(* Logix 5000 project; controller NSH_PLC2 vendor 1 type 14 code 167 rev 32.14; software revision 32.03; part 4 of 6 *)
(* tags used below, declared in another part *)
   AOI_MCC3_10J_ToPLC1 : E300ToMotor;
   AOI_MCC3_11A_ToPLC1 : E300ToMotor;
   AOI_MCC3_11D_ToPLC1 : E300ToMotor;
   AOI_MCC3_11G_ToPLC1 : E300ToMotor;
   AOI_MCC3_11J_ToPLC1 : E300ToMotor;
   AOI_MCC3_12A_ToPLC1 : E300ToMotor;
   AOI_MCC3_12C_ToPLC1 : E300ToMotor;
   AOI_MCC3_12E_ToPLC1 : E300ToMotor;
   AOI_MCC3_12G_ToPLC1 : E300ToMotor;
   AOI_MCC3_12J_ToPLC1 : E300ToMotor;
   AOI_MCC3_12L_ToPLC1 : E300ToMotor;
   AOI_MCC3_13A_ToPLC1 : E300ToMotor;
   AOI_MCC3_13C_ToPLC1 : E300ToMotor;
   AOI_MCC3_13E_ToPLC1 : E300ToMotor;
   AOI_MCC3_13G_ToPLC1 : E300ToMotor;
   AOI_MCC3_13J_ToPLC1 : E300ToMotor;
   AOI_MCC3_13L_ToPLC1 : E300ToMotor;
   AOI_MCC3_14A_ToPLC1 : E300ToMotor;
   AOI_MCC3_14C_ToPLC1 : E300ToMotor;
   AOI_MCC3_14E_ToPLC1 : E300ToMotor;
   AOI_MCC3_14G_ToPLC1 : E300ToMotor;
   AOI_MCC3_14J_ToPLC1 : E300ToMotor;
   AOI_MCC3_14L_ToPLC1 : E300ToMotor;
   AOI_MCC3_15A_ToPLC1 : E300ToMotor;
   AOI_MCC3_15C_ToPLC1 : E300ToMotor;
   AOI_MCC3_15E_ToPLC1 : E300ToMotor;
   AOI_MCC3_15G_ToPLC1 : E300ToMotor;
   AOI_MCC3_15J_ToPLC1 : E300ToMotor;
   AOI_MCC3_16A_ToPLC1 : E300ToMotor;
   AOI_MCC3_16C_ToPLC1 : E300ToMotor;
   AOI_MCC3_16E_ToPLC1 : E300ToMotor;
   AOI_MCC3_16G_ToPLC1 : E300ToMotor;
   AOI_MCC3_16J_ToPLC1 : E300ToMotor;
   AOI_MCC3_16L_ToPLC1 : E300ToMotor;
   AOI_MCC3_17A_ToPLC1 : E300ToMotor;
   AOI_MCC3_17C_ToPLC1 : E300ToMotor;
   AOI_MCC3_17E_ToPLC1 : E300ToMotor;
   AOI_MCC3_17G_ToPLC1 : E300ToMotor;
   AOI_MCC3_17J_ToPLC1 : E300ToMotor;
   AOI_MCC3_17L_ToPLC1 : E300ToMotor;
   AOI_MCC3_18A_ToPLC1 : E300ToMotor;
   AOI_MCC3_18C_ToPLC1 : E300ToMotor;
   AOI_MCC3_18E_ToPLC1 : E300ToMotor;
   AOI_MCC3_18G_ToPLC1 : E300ToMotor;
   AOI_MCC3_18J_ToPLC1 : E300ToMotor;
   AOI_MCC3_18L_ToPLC1 : E300ToMotor;
   AOI_MCC3_19A_ToPLC1 : E300ToMotor;
   AOI_MCC3_19C_ToPLC1 : E300ToMotor;
   AOI_MCC3_19E_ToPLC1 : E300ToMotor;
   AOI_MCC3_19G_ToPLC1 : E300ToMotor;
   AOI_MCC3_19J_ToPLC1 : E300ToMotor;
   AOI_MCC3_20A_ToPLC1 : E300ToMotor;
   AOI_MCC3_20C_ToPLC1 : E300ToMotor;
   AOI_MCC3_20E_ToPLC1 : E300ToMotor;
   AOI_MCC3_20G_ToPLC1 : E300ToMotor;
   AOI_MCC3_20J_ToPLC1 : E300ToMotor;
   AOI_MCC3_21A_ToPLC1 : E300ToMotor;
   AOI_MCC3_21C_ToPLC1 : E300ToMotor;
   AOI_MCC3_21E_ToPLC1 : E300ToMotor;
   AOI_MCC3_21G_ToPLC1 : E300ToMotor;
   AOI_MCC3_21J_ToPLC1 : E300ToMotor;
   AOI_MCC3_21L_ToPLC1 : E300ToMotor;
   AOI_MCC3_22C_ToPLC1 : E300ToMotor;
   AOI_MCC3_22E_ToPLC1 : E300ToMotor;
   AOI_MCC4_1E_ToPLC1 : PF525ToMotor;
   AOI_MCC4_2A_ToPLC1 : E300ToMotor;
   AOI_MCC4_2C_ToPLC1 : E300ToMotor;
   AOI_MCC4_2E_ToPLC1 : E300ToMotor;
   AOI_MCC4_2G_ToPLC1 : PF525ToMotor;
   AOI_MCC4_2K_ToPLC1 : PF525ToMotor;
   AOI_MCC4_3A_ToPLC1 : E300ToMotor;
   AOI_MCC4_3C_ToPLC1 : E300ToMotor;
   Const_4000_Hex : INT;   // Constant #16:4000, Entry Status Communicating
   GSV_EntryStatus : INT;   // GSV Entry Status, shold be #16:4000
   MCC3_10J_CommsOK : BOOL;   // Communications with AOP OK
   MCC3_11A_CommsOK : BOOL;   // Communications with AOP OK
   MCC3_11D_CommsOK : BOOL;   // Communications with AOP OK
   MCC3_11G_CommsOK : BOOL;   // Communications with AOP OK
   MCC3_11J_CommsOK : BOOL;   // Communications with AOP OK
   MCC3_12A_CommsOK : BOOL;   // Communications with AOP OK
   MCC3_12C_CommsOK : BOOL;   // Communications with AOP OK
   MCC3_12E_CommsOK : BOOL;   // Communications with AOP OK
   MCC3_12G_CommsOK : BOOL;   // Communications with AOP OK
   MCC3_12J_CommsOK : BOOL;   // Communications with AOP OK
   MCC3_12L_CommsOK : BOOL;   // Communications with AOP OK
   MCC3_13A_CommsOK : BOOL;   // Communications with AOP OK
   MCC3_13C_CommsOK : BOOL;   // Communications with AOP OK
   MCC3_13E_CommsOK : BOOL;   // Communications with AOP OK
   MCC3_13G_CommsOK : BOOL;   // Communications with AOP OK
   MCC3_13J_CommsOK : BOOL;   // Communications with AOP OK
   MCC3_13L_CommsOK : BOOL;   // Communications with AOP OK
   MCC3_14A_CommsOK : BOOL;   // Communications with AOP OK
   MCC3_14C_CommsOK : BOOL;   // Communications with AOP OK
   MCC3_14E_CommsOK : BOOL;   // Communications with AOP OK
   MCC3_14G_CommsOK : BOOL;   // Communications with AOP OK
   MCC3_14J_CommsOK : BOOL;   // Communications with AOP OK
   MCC3_14L_CommsOK : BOOL;   // Communications with AOP OK
   MCC3_15A_CommsOK : BOOL;   // Communications with AOP OK
   MCC3_15C_CommsOK : BOOL;   // Communications with AOP OK
   MCC3_15E_CommsOK : BOOL;   // Communications with AOP OK
   MCC3_15G_CommsOK : BOOL;   // Communications with AOP OK
   MCC3_15J_CommsOK : BOOL;   // Communications with AOP OK
   MCC3_16A_CommsOK : BOOL;   // Communications with AOP OK
   MCC3_16C_CommsOK : BOOL;   // Communications with AOP OK
   MCC3_16E_CommsOK : BOOL;   // Communications with AOP OK
   MCC3_16G_CommsOK : BOOL;   // Communications with AOP OK
   MCC3_16J_CommsOK : BOOL;   // Communications with AOP OK
   MCC3_16L_CommsOK : BOOL;   // Communications with AOP OK
   MCC3_17A_CommsOK : BOOL;   // Communications with AOP OK
   MCC3_17C_CommsOK : BOOL;   // Communications with AOP OK
   MCC3_17E_CommsOK : BOOL;   // Communications with AOP OK
   MCC3_17G_CommsOK : BOOL;   // Communications with AOP OK
   MCC3_17J_CommsOK : BOOL;   // Communications with AOP OK
   MCC3_17L_CommsOK : BOOL;   // Communications with AOP OK
   MCC3_18A_CommsOK : BOOL;   // Communications with AOP OK
   MCC3_18C_CommsOK : BOOL;   // Communications with AOP OK
   MCC3_18E_CommsOK : BOOL;   // Communications with AOP OK
   MCC3_18G_CommsOK : BOOL;   // Communications with AOP OK
   MCC3_18J_CommsOK : BOOL;   // Communications with AOP OK
   MCC3_18L_CommsOK : BOOL;   // Communications with AOP OK
   MCC3_19A_CommsOK : BOOL;   // Communications with AOP OK
   MCC3_19C_CommsOK : BOOL;   // Communications with AOP OK
   MCC3_19E_CommsOK : BOOL;   // Communications with AOP OK
   MCC3_19G_CommsOK : BOOL;   // Communications with AOP OK
   MCC3_19J_CommsOK : BOOL;   // Communications with AOP OK
   MCC3_20A_CommsOK : BOOL;   // Communications with AOP OK
   MCC3_20C_CommsOK : BOOL;   // Communications with AOP OK
   MCC3_20E_CommsOK : BOOL;   // Communications with AOP OK
   MCC3_20G_CommsOK : BOOL;   // Communications with AOP OK
   MCC3_20J_CommsOK : BOOL;   // Communications with AOP OK
   MCC3_21A_CommsOK : BOOL;   // Communications with AOP OK
   MCC3_21C_CommsOK : BOOL;   // Communications with AOP OK
   MCC3_21E_CommsOK : BOOL;   // Communications with AOP OK
   MCC3_21G_CommsOK : BOOL;   // Communications with AOP OK
   MCC3_21J_CommsOK : BOOL;   // Communications with AOP OK
   MCC3_21L_CommsOK : BOOL;   // Communications with AOP OK
   MCC3_22C_CommsOK : BOOL;   // Communications with AOP OK
   MCC3_22E_CommsOK : BOOL;   // Communications with AOP OK
   MCC4_1E_CommsOK : BOOL;   // Communications with AOP OK
   MCC4_2A_CommsOK : BOOL;   // Communications with AOP OK
   MCC4_2C_CommsOK : BOOL;   // Communications with AOP OK
   MCC4_2E_CommsOK : BOOL;   // Communications with AOP OK
   MCC4_2G_CommsOK : BOOL;   // Communications with AOP OK
   MCC4_2K_CommsOK : BOOL;   // Communications with AOP OK
   MCC4_3A_CommsOK : BOOL;   // Communications with AOP OK
   MCC4_3C_CommsOK : BOOL;   // Communications with AOP OK
   MotorsStatusTag : MotorsStatusUDT;   // Only Instance of UDT
(* MainProgram, continued *)

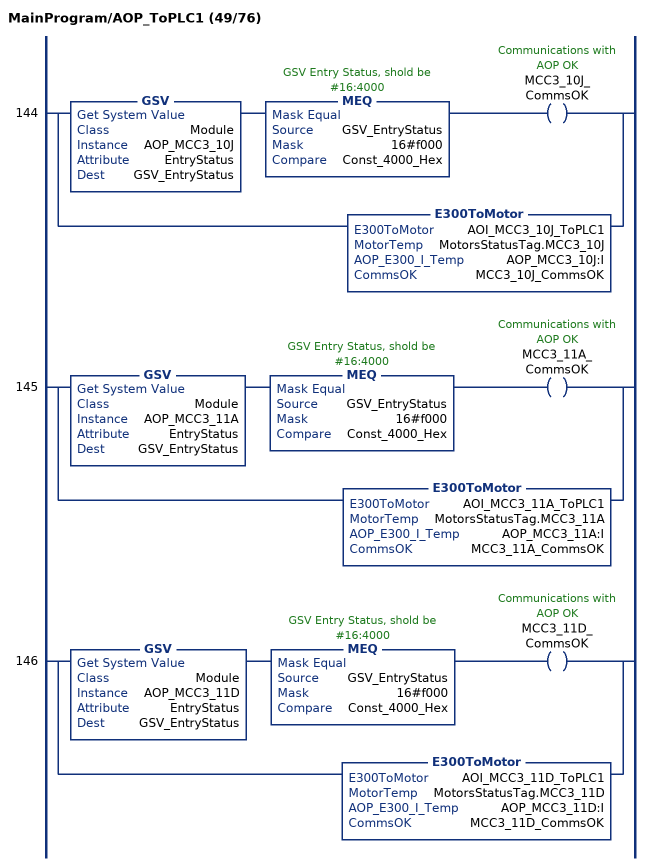
   [picture p55: MainProgram/AOP_ToPLC1 rungs 144-146]
   144: [GSV(Module,AOP_MCC3_10J,EntryStatus,GSV_EntryStatus) MEQ(GSV_EntryStatus,16#f000,Const_4000_Hex) OTE(MCC3_10J_CommsOK) ,E300ToMotor(AOI_MCC3_10J_ToPLC1,MotorsStatusTag.MCC3_10J,AOP_MCC3_10J:I,MCC3_10J_CommsOK) ];
   145: [GSV(Module,AOP_MCC3_11A,EntryStatus,GSV_EntryStatus) MEQ(GSV_EntryStatus,16#f000,Const_4000_Hex) OTE(MCC3_11A_CommsOK) ,E300ToMotor(AOI_MCC3_11A_ToPLC1,MotorsStatusTag.MCC3_11A,AOP_MCC3_11A:I,MCC3_11A_CommsOK) ];
   146: [GSV(Module,AOP_MCC3_11D,EntryStatus,GSV_EntryStatus) MEQ(GSV_EntryStatus,16#f000,Const_4000_Hex) OTE(MCC3_11D_CommsOK) ,E300ToMotor(AOI_MCC3_11D_ToPLC1,MotorsStatusTag.MCC3_11D,AOP_MCC3_11D:I,MCC3_11D_CommsOK) ];
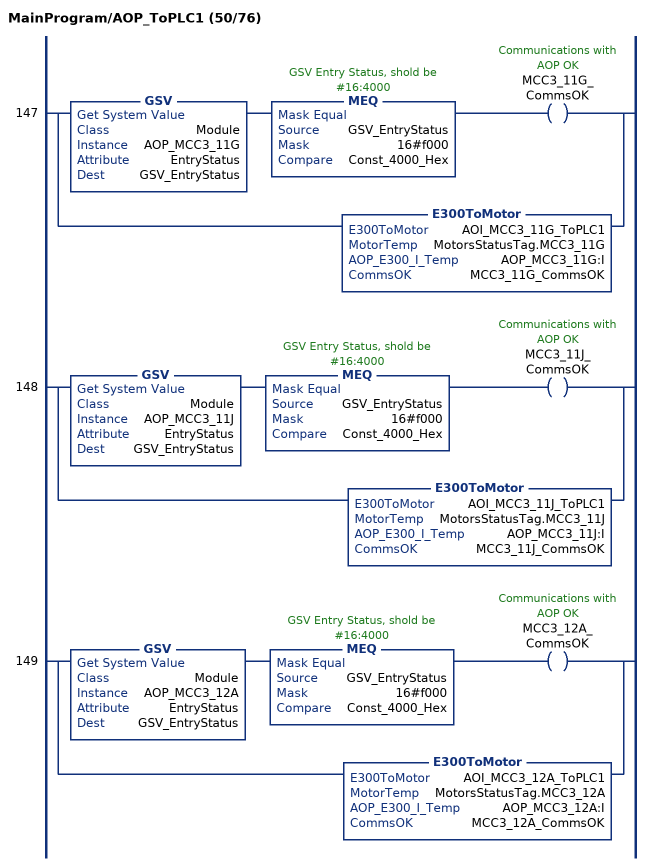
   147: [GSV(Module,AOP_MCC3_11G,EntryStatus,GSV_EntryStatus) MEQ(GSV_EntryStatus,16#f000,Const_4000_Hex) OTE(MCC3_11G_CommsOK) ,E300ToMotor(AOI_MCC3_11G_ToPLC1,MotorsStatusTag.MCC3_11G,AOP_MCC3_11G:I,MCC3_11G_CommsOK) ];
   148: [GSV(Module,AOP_MCC3_11J,EntryStatus,GSV_EntryStatus) MEQ(GSV_EntryStatus,16#f000,Const_4000_Hex) OTE(MCC3_11J_CommsOK) ,E300ToMotor(AOI_MCC3_11J_ToPLC1,MotorsStatusTag.MCC3_11J,AOP_MCC3_11J:I,MCC3_11J_CommsOK) ];
   149: [GSV(Module,AOP_MCC3_12A,EntryStatus,GSV_EntryStatus) MEQ(GSV_EntryStatus,16#f000,Const_4000_Hex) OTE(MCC3_12A_CommsOK) ,E300ToMotor(AOI_MCC3_12A_ToPLC1,MotorsStatusTag.MCC3_12A,AOP_MCC3_12A:I,MCC3_12A_CommsOK) ];
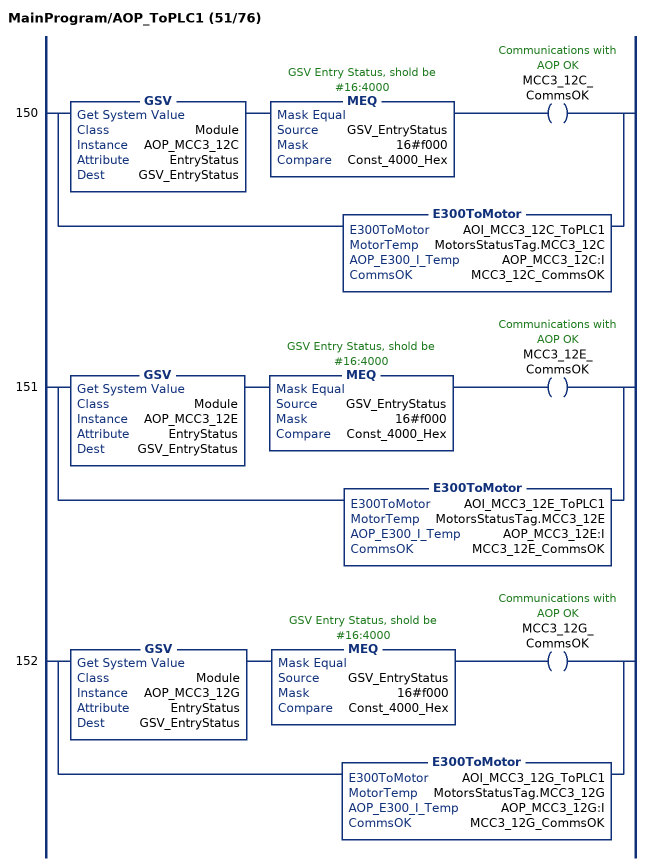
   150: [GSV(Module,AOP_MCC3_12C,EntryStatus,GSV_EntryStatus) MEQ(GSV_EntryStatus,16#f000,Const_4000_Hex) OTE(MCC3_12C_CommsOK) ,E300ToMotor(AOI_MCC3_12C_ToPLC1,MotorsStatusTag.MCC3_12C,AOP_MCC3_12C:I,MCC3_12C_CommsOK) ];
   151: [GSV(Module,AOP_MCC3_12E,EntryStatus,GSV_EntryStatus) MEQ(GSV_EntryStatus,16#f000,Const_4000_Hex) OTE(MCC3_12E_CommsOK) ,E300ToMotor(AOI_MCC3_12E_ToPLC1,MotorsStatusTag.MCC3_12E,AOP_MCC3_12E:I,MCC3_12E_CommsOK) ];
   152: [GSV(Module,AOP_MCC3_12G,EntryStatus,GSV_EntryStatus) MEQ(GSV_EntryStatus,16#f000,Const_4000_Hex) OTE(MCC3_12G_CommsOK) ,E300ToMotor(AOI_MCC3_12G_ToPLC1,MotorsStatusTag.MCC3_12G,AOP_MCC3_12G:I,MCC3_12G_CommsOK) ];
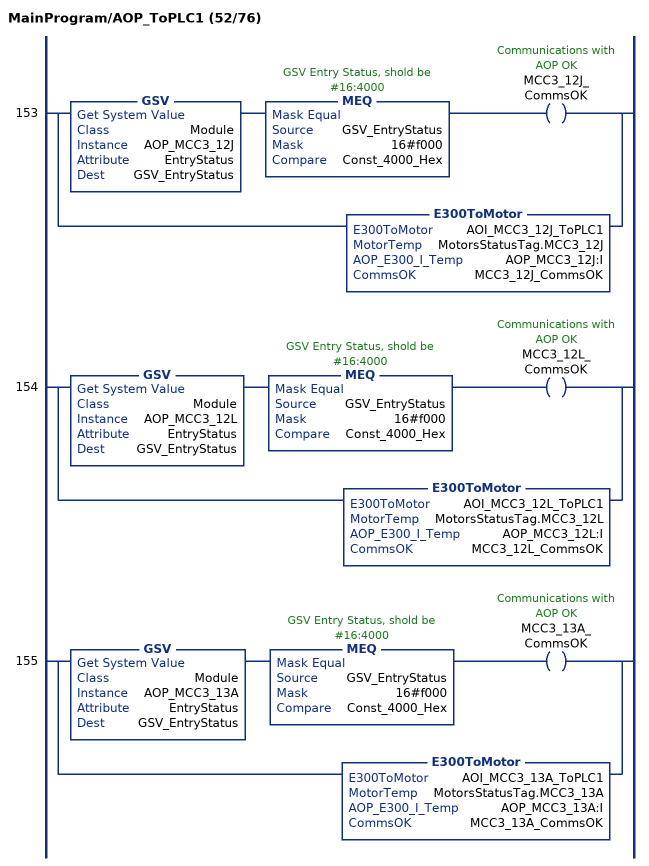
   153: [GSV(Module,AOP_MCC3_12J,EntryStatus,GSV_EntryStatus) MEQ(GSV_EntryStatus,16#f000,Const_4000_Hex) OTE(MCC3_12J_CommsOK) ,E300ToMotor(AOI_MCC3_12J_ToPLC1,MotorsStatusTag.MCC3_12J,AOP_MCC3_12J:I,MCC3_12J_CommsOK) ];
   154: [GSV(Module,AOP_MCC3_12L,EntryStatus,GSV_EntryStatus) MEQ(GSV_EntryStatus,16#f000,Const_4000_Hex) OTE(MCC3_12L_CommsOK) ,E300ToMotor(AOI_MCC3_12L_ToPLC1,MotorsStatusTag.MCC3_12L,AOP_MCC3_12L:I,MCC3_12L_CommsOK) ];
   155: [GSV(Module,AOP_MCC3_13A,EntryStatus,GSV_EntryStatus) MEQ(GSV_EntryStatus,16#f000,Const_4000_Hex) OTE(MCC3_13A_CommsOK) ,E300ToMotor(AOI_MCC3_13A_ToPLC1,MotorsStatusTag.MCC3_13A,AOP_MCC3_13A:I,MCC3_13A_CommsOK) ];
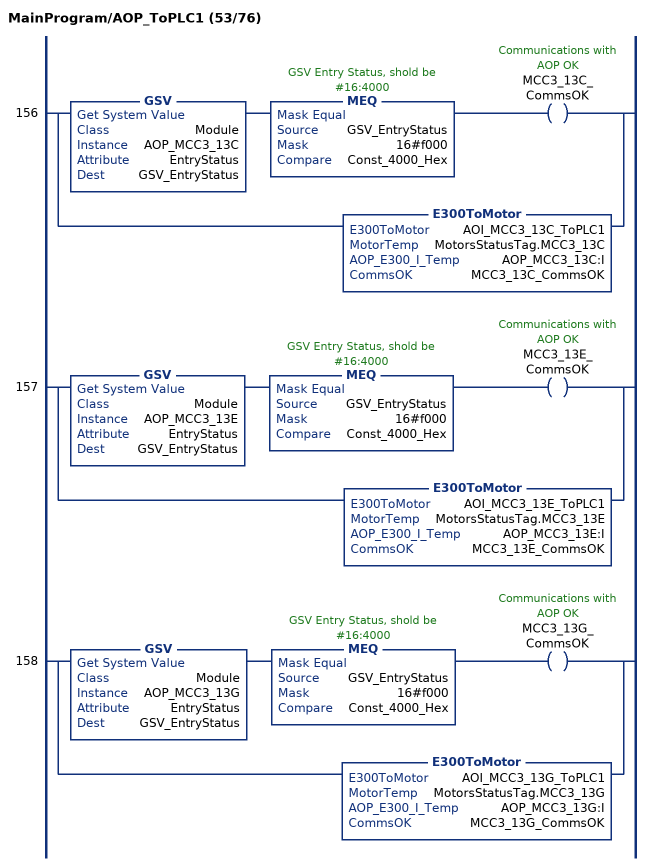
   156: [GSV(Module,AOP_MCC3_13C,EntryStatus,GSV_EntryStatus) MEQ(GSV_EntryStatus,16#f000,Const_4000_Hex) OTE(MCC3_13C_CommsOK) ,E300ToMotor(AOI_MCC3_13C_ToPLC1,MotorsStatusTag.MCC3_13C,AOP_MCC3_13C:I,MCC3_13C_CommsOK) ];
   157: [GSV(Module,AOP_MCC3_13E,EntryStatus,GSV_EntryStatus) MEQ(GSV_EntryStatus,16#f000,Const_4000_Hex) OTE(MCC3_13E_CommsOK) ,E300ToMotor(AOI_MCC3_13E_ToPLC1,MotorsStatusTag.MCC3_13E,AOP_MCC3_13E:I,MCC3_13E_CommsOK) ];
   158: [GSV(Module,AOP_MCC3_13G,EntryStatus,GSV_EntryStatus) MEQ(GSV_EntryStatus,16#f000,Const_4000_Hex) OTE(MCC3_13G_CommsOK) ,E300ToMotor(AOI_MCC3_13G_ToPLC1,MotorsStatusTag.MCC3_13G,AOP_MCC3_13G:I,MCC3_13G_CommsOK) ];
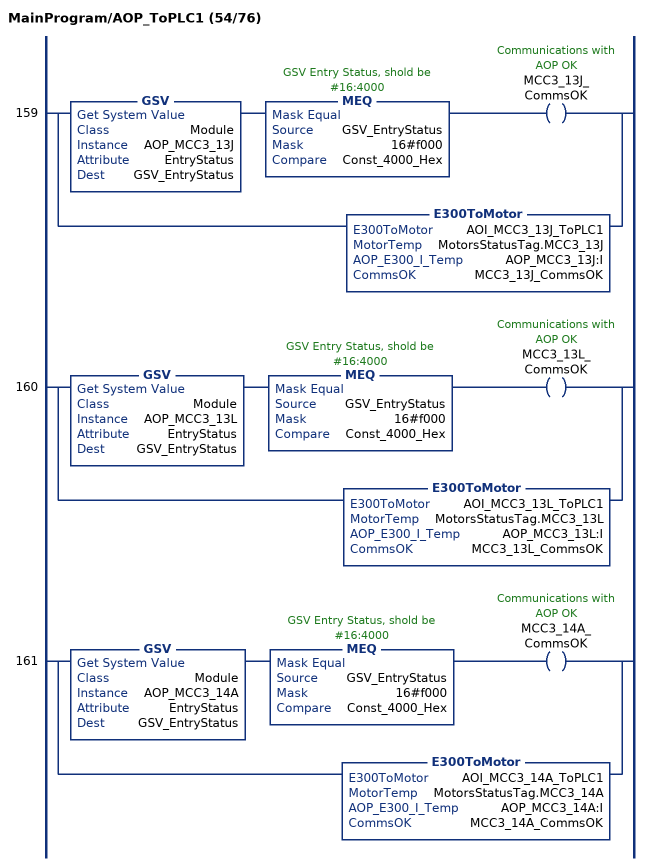
   159: [GSV(Module,AOP_MCC3_13J,EntryStatus,GSV_EntryStatus) MEQ(GSV_EntryStatus,16#f000,Const_4000_Hex) OTE(MCC3_13J_CommsOK) ,E300ToMotor(AOI_MCC3_13J_ToPLC1,MotorsStatusTag.MCC3_13J,AOP_MCC3_13J:I,MCC3_13J_CommsOK) ];
   160: [GSV(Module,AOP_MCC3_13L,EntryStatus,GSV_EntryStatus) MEQ(GSV_EntryStatus,16#f000,Const_4000_Hex) OTE(MCC3_13L_CommsOK) ,E300ToMotor(AOI_MCC3_13L_ToPLC1,MotorsStatusTag.MCC3_13L,AOP_MCC3_13L:I,MCC3_13L_CommsOK) ];
   161: [GSV(Module,AOP_MCC3_14A,EntryStatus,GSV_EntryStatus) MEQ(GSV_EntryStatus,16#f000,Const_4000_Hex) OTE(MCC3_14A_CommsOK) ,E300ToMotor(AOI_MCC3_14A_ToPLC1,MotorsStatusTag.MCC3_14A,AOP_MCC3_14A:I,MCC3_14A_CommsOK) ];
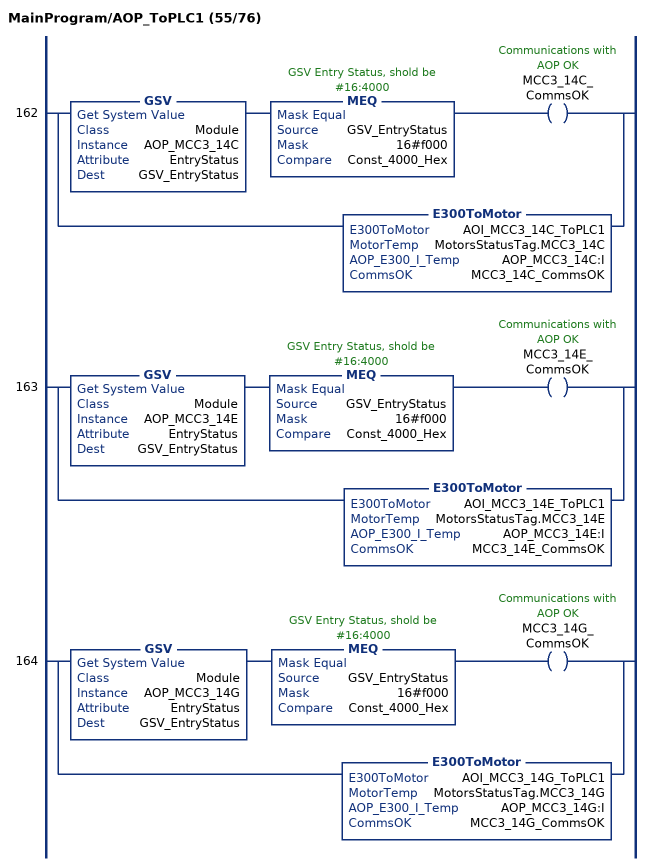
   162: [GSV(Module,AOP_MCC3_14C,EntryStatus,GSV_EntryStatus) MEQ(GSV_EntryStatus,16#f000,Const_4000_Hex) OTE(MCC3_14C_CommsOK) ,E300ToMotor(AOI_MCC3_14C_ToPLC1,MotorsStatusTag.MCC3_14C,AOP_MCC3_14C:I,MCC3_14C_CommsOK) ];
   163: [GSV(Module,AOP_MCC3_14E,EntryStatus,GSV_EntryStatus) MEQ(GSV_EntryStatus,16#f000,Const_4000_Hex) OTE(MCC3_14E_CommsOK) ,E300ToMotor(AOI_MCC3_14E_ToPLC1,MotorsStatusTag.MCC3_14E,AOP_MCC3_14E:I,MCC3_14E_CommsOK) ];
   164: [GSV(Module,AOP_MCC3_14G,EntryStatus,GSV_EntryStatus) MEQ(GSV_EntryStatus,16#f000,Const_4000_Hex) OTE(MCC3_14G_CommsOK) ,E300ToMotor(AOI_MCC3_14G_ToPLC1,MotorsStatusTag.MCC3_14G,AOP_MCC3_14G:I,MCC3_14G_CommsOK) ];
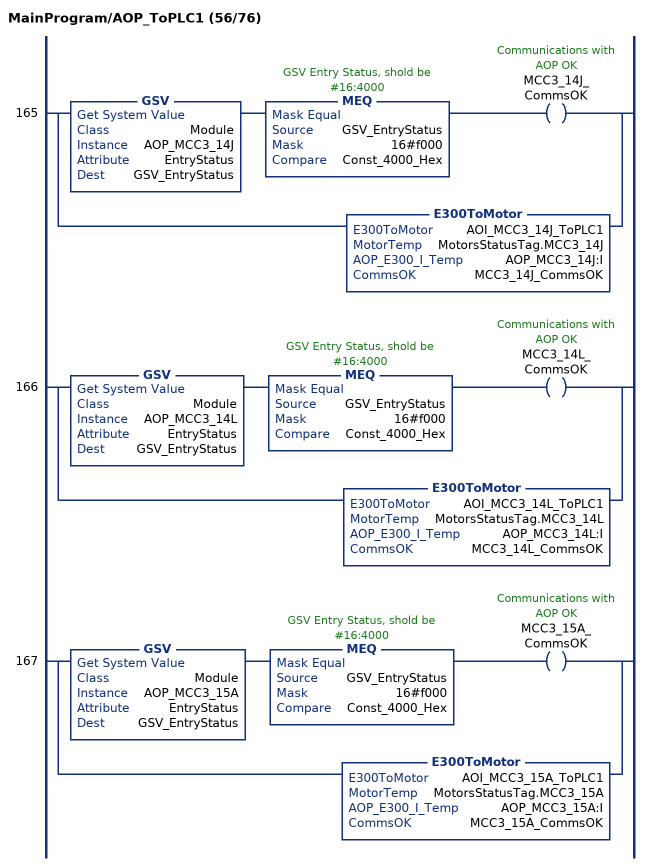
   165: [GSV(Module,AOP_MCC3_14J,EntryStatus,GSV_EntryStatus) MEQ(GSV_EntryStatus,16#f000,Const_4000_Hex) OTE(MCC3_14J_CommsOK) ,E300ToMotor(AOI_MCC3_14J_ToPLC1,MotorsStatusTag.MCC3_14J,AOP_MCC3_14J:I,MCC3_14J_CommsOK) ];
   166: [GSV(Module,AOP_MCC3_14L,EntryStatus,GSV_EntryStatus) MEQ(GSV_EntryStatus,16#f000,Const_4000_Hex) OTE(MCC3_14L_CommsOK) ,E300ToMotor(AOI_MCC3_14L_ToPLC1,MotorsStatusTag.MCC3_14L,AOP_MCC3_14L:I,MCC3_14L_CommsOK) ];
   167: [GSV(Module,AOP_MCC3_15A,EntryStatus,GSV_EntryStatus) MEQ(GSV_EntryStatus,16#f000,Const_4000_Hex) OTE(MCC3_15A_CommsOK) ,E300ToMotor(AOI_MCC3_15A_ToPLC1,MotorsStatusTag.MCC3_15A,AOP_MCC3_15A:I,MCC3_15A_CommsOK) ];
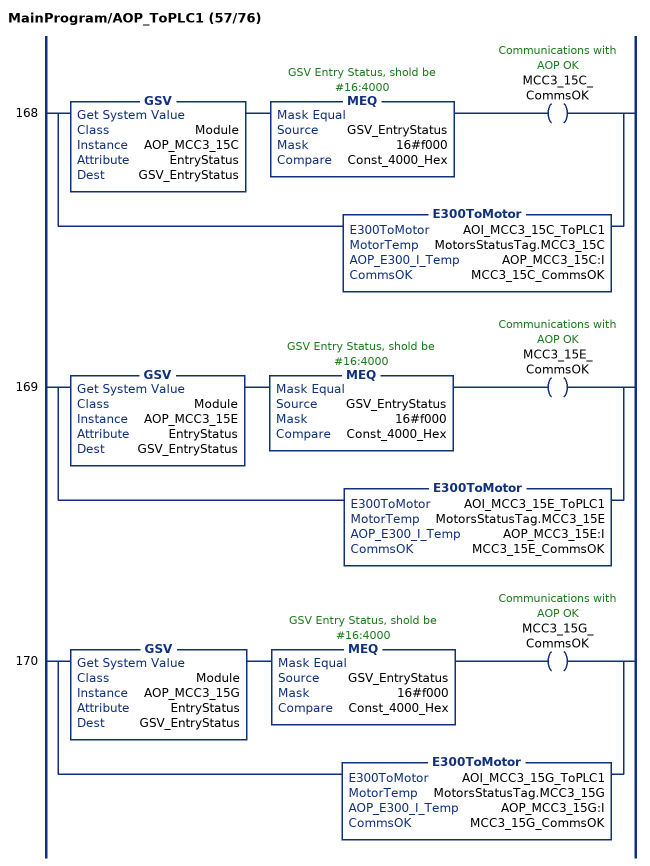
   168: [GSV(Module,AOP_MCC3_15C,EntryStatus,GSV_EntryStatus) MEQ(GSV_EntryStatus,16#f000,Const_4000_Hex) OTE(MCC3_15C_CommsOK) ,E300ToMotor(AOI_MCC3_15C_ToPLC1,MotorsStatusTag.MCC3_15C,AOP_MCC3_15C:I,MCC3_15C_CommsOK) ];
   169: [GSV(Module,AOP_MCC3_15E,EntryStatus,GSV_EntryStatus) MEQ(GSV_EntryStatus,16#f000,Const_4000_Hex) OTE(MCC3_15E_CommsOK) ,E300ToMotor(AOI_MCC3_15E_ToPLC1,MotorsStatusTag.MCC3_15E,AOP_MCC3_15E:I,MCC3_15E_CommsOK) ];
   170: [GSV(Module,AOP_MCC3_15G,EntryStatus,GSV_EntryStatus) MEQ(GSV_EntryStatus,16#f000,Const_4000_Hex) OTE(MCC3_15G_CommsOK) ,E300ToMotor(AOI_MCC3_15G_ToPLC1,MotorsStatusTag.MCC3_15G,AOP_MCC3_15G:I,MCC3_15G_CommsOK) ];
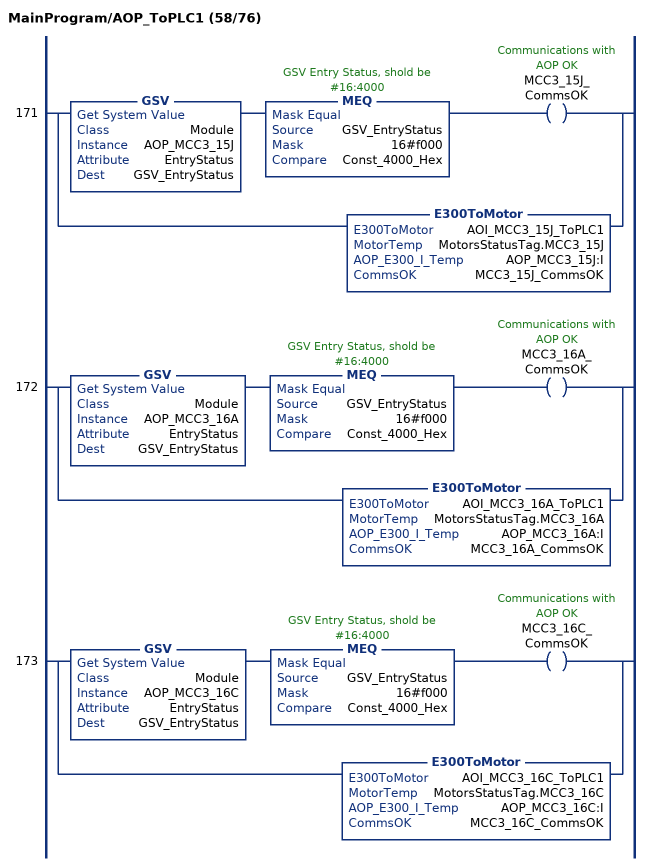
   171: [GSV(Module,AOP_MCC3_15J,EntryStatus,GSV_EntryStatus) MEQ(GSV_EntryStatus,16#f000,Const_4000_Hex) OTE(MCC3_15J_CommsOK) ,E300ToMotor(AOI_MCC3_15J_ToPLC1,MotorsStatusTag.MCC3_15J,AOP_MCC3_15J:I,MCC3_15J_CommsOK) ];
   172: [GSV(Module,AOP_MCC3_16A,EntryStatus,GSV_EntryStatus) MEQ(GSV_EntryStatus,16#f000,Const_4000_Hex) OTE(MCC3_16A_CommsOK) ,E300ToMotor(AOI_MCC3_16A_ToPLC1,MotorsStatusTag.MCC3_16A,AOP_MCC3_16A:I,MCC3_16A_CommsOK) ];
   173: [GSV(Module,AOP_MCC3_16C,EntryStatus,GSV_EntryStatus) MEQ(GSV_EntryStatus,16#f000,Const_4000_Hex) OTE(MCC3_16C_CommsOK) ,E300ToMotor(AOI_MCC3_16C_ToPLC1,MotorsStatusTag.MCC3_16C,AOP_MCC3_16C:I,MCC3_16C_CommsOK) ];
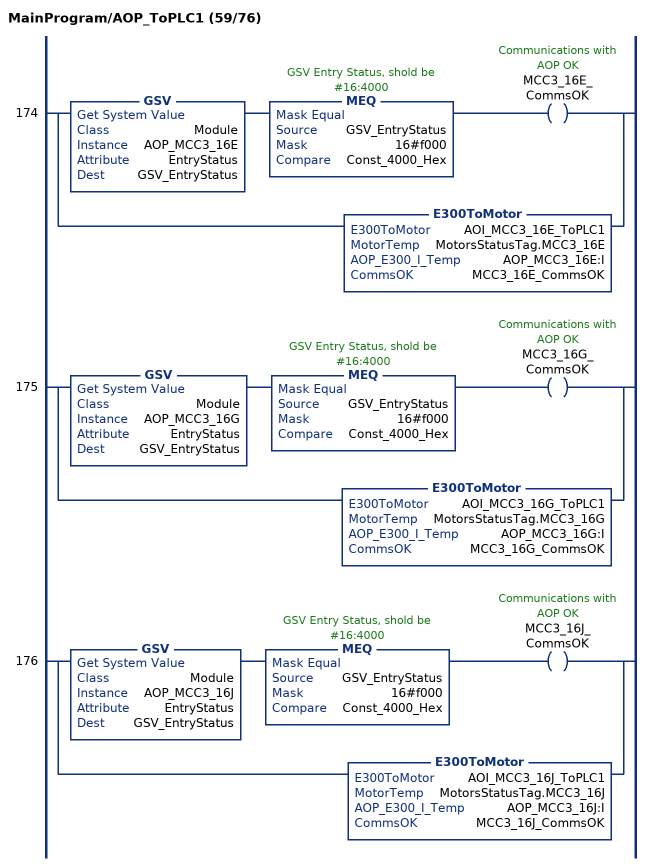
   174: [GSV(Module,AOP_MCC3_16E,EntryStatus,GSV_EntryStatus) MEQ(GSV_EntryStatus,16#f000,Const_4000_Hex) OTE(MCC3_16E_CommsOK) ,E300ToMotor(AOI_MCC3_16E_ToPLC1,MotorsStatusTag.MCC3_16E,AOP_MCC3_16E:I,MCC3_16E_CommsOK) ];
   175: [GSV(Module,AOP_MCC3_16G,EntryStatus,GSV_EntryStatus) MEQ(GSV_EntryStatus,16#f000,Const_4000_Hex) OTE(MCC3_16G_CommsOK) ,E300ToMotor(AOI_MCC3_16G_ToPLC1,MotorsStatusTag.MCC3_16G,AOP_MCC3_16G:I,MCC3_16G_CommsOK) ];
   176: [GSV(Module,AOP_MCC3_16J,EntryStatus,GSV_EntryStatus) MEQ(GSV_EntryStatus,16#f000,Const_4000_Hex) OTE(MCC3_16J_CommsOK) ,E300ToMotor(AOI_MCC3_16J_ToPLC1,MotorsStatusTag.MCC3_16J,AOP_MCC3_16J:I,MCC3_16J_CommsOK) ];
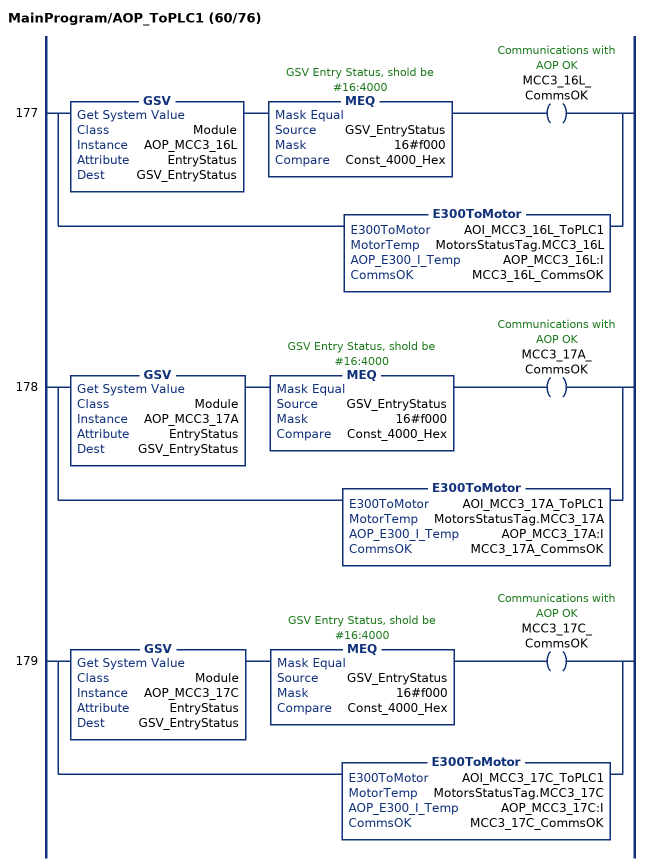
   177: [GSV(Module,AOP_MCC3_16L,EntryStatus,GSV_EntryStatus) MEQ(GSV_EntryStatus,16#f000,Const_4000_Hex) OTE(MCC3_16L_CommsOK) ,E300ToMotor(AOI_MCC3_16L_ToPLC1,MotorsStatusTag.MCC3_16L,AOP_MCC3_16L:I,MCC3_16L_CommsOK) ];
   178: [GSV(Module,AOP_MCC3_17A,EntryStatus,GSV_EntryStatus) MEQ(GSV_EntryStatus,16#f000,Const_4000_Hex) OTE(MCC3_17A_CommsOK) ,E300ToMotor(AOI_MCC3_17A_ToPLC1,MotorsStatusTag.MCC3_17A,AOP_MCC3_17A:I,MCC3_17A_CommsOK) ];
   179: [GSV(Module,AOP_MCC3_17C,EntryStatus,GSV_EntryStatus) MEQ(GSV_EntryStatus,16#f000,Const_4000_Hex) OTE(MCC3_17C_CommsOK) ,E300ToMotor(AOI_MCC3_17C_ToPLC1,MotorsStatusTag.MCC3_17C,AOP_MCC3_17C:I,MCC3_17C_CommsOK) ];
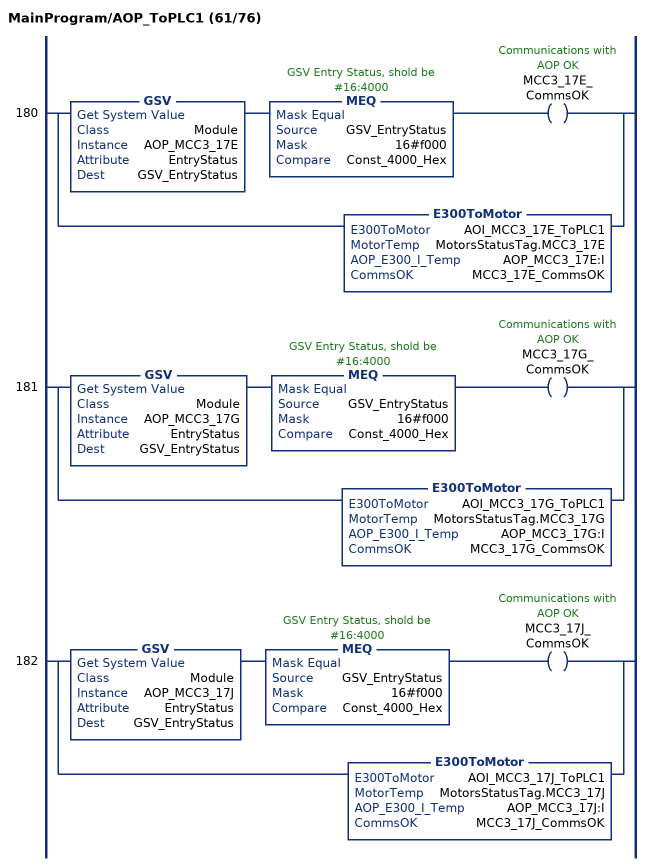
   180: [GSV(Module,AOP_MCC3_17E,EntryStatus,GSV_EntryStatus) MEQ(GSV_EntryStatus,16#f000,Const_4000_Hex) OTE(MCC3_17E_CommsOK) ,E300ToMotor(AOI_MCC3_17E_ToPLC1,MotorsStatusTag.MCC3_17E,AOP_MCC3_17E:I,MCC3_17E_CommsOK) ];
   181: [GSV(Module,AOP_MCC3_17G,EntryStatus,GSV_EntryStatus) MEQ(GSV_EntryStatus,16#f000,Const_4000_Hex) OTE(MCC3_17G_CommsOK) ,E300ToMotor(AOI_MCC3_17G_ToPLC1,MotorsStatusTag.MCC3_17G,AOP_MCC3_17G:I,MCC3_17G_CommsOK) ];
   182: [GSV(Module,AOP_MCC3_17J,EntryStatus,GSV_EntryStatus) MEQ(GSV_EntryStatus,16#f000,Const_4000_Hex) OTE(MCC3_17J_CommsOK) ,E300ToMotor(AOI_MCC3_17J_ToPLC1,MotorsStatusTag.MCC3_17J,AOP_MCC3_17J:I,MCC3_17J_CommsOK) ];
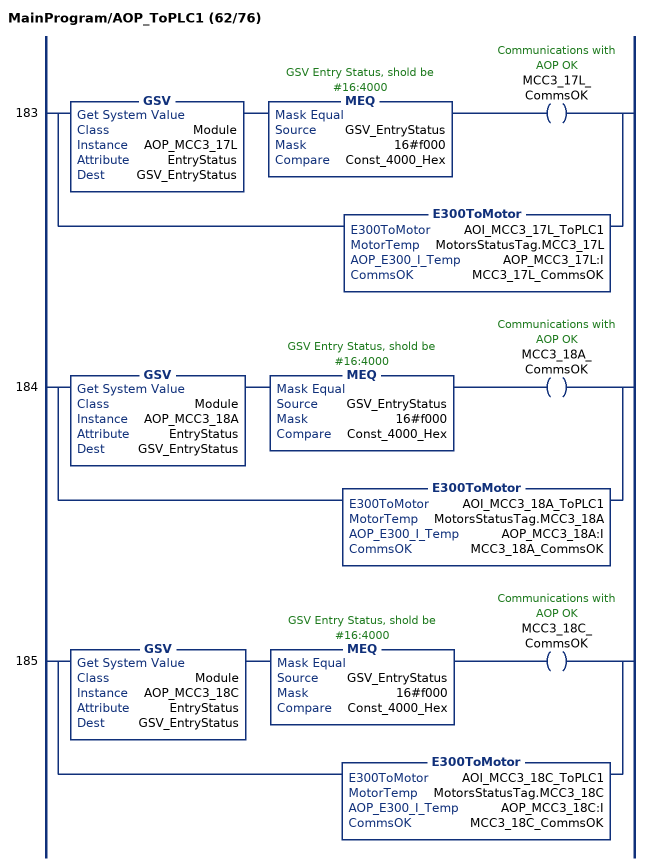
   183: [GSV(Module,AOP_MCC3_17L,EntryStatus,GSV_EntryStatus) MEQ(GSV_EntryStatus,16#f000,Const_4000_Hex) OTE(MCC3_17L_CommsOK) ,E300ToMotor(AOI_MCC3_17L_ToPLC1,MotorsStatusTag.MCC3_17L,AOP_MCC3_17L:I,MCC3_17L_CommsOK) ];
   184: [GSV(Module,AOP_MCC3_18A,EntryStatus,GSV_EntryStatus) MEQ(GSV_EntryStatus,16#f000,Const_4000_Hex) OTE(MCC3_18A_CommsOK) ,E300ToMotor(AOI_MCC3_18A_ToPLC1,MotorsStatusTag.MCC3_18A,AOP_MCC3_18A:I,MCC3_18A_CommsOK) ];
   185: [GSV(Module,AOP_MCC3_18C,EntryStatus,GSV_EntryStatus) MEQ(GSV_EntryStatus,16#f000,Const_4000_Hex) OTE(MCC3_18C_CommsOK) ,E300ToMotor(AOI_MCC3_18C_ToPLC1,MotorsStatusTag.MCC3_18C,AOP_MCC3_18C:I,MCC3_18C_CommsOK) ];
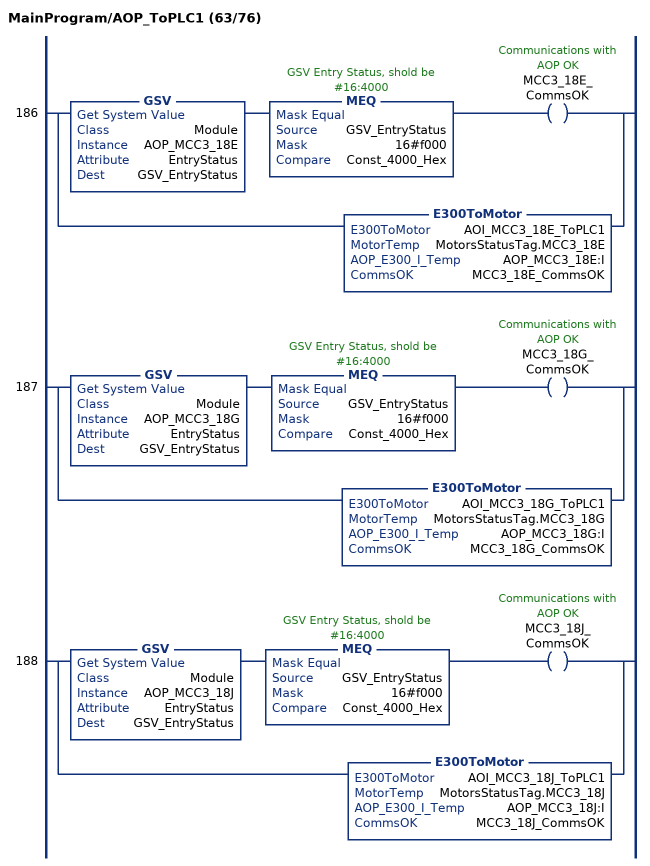
   186: [GSV(Module,AOP_MCC3_18E,EntryStatus,GSV_EntryStatus) MEQ(GSV_EntryStatus,16#f000,Const_4000_Hex) OTE(MCC3_18E_CommsOK) ,E300ToMotor(AOI_MCC3_18E_ToPLC1,MotorsStatusTag.MCC3_18E,AOP_MCC3_18E:I,MCC3_18E_CommsOK) ];
   187: [GSV(Module,AOP_MCC3_18G,EntryStatus,GSV_EntryStatus) MEQ(GSV_EntryStatus,16#f000,Const_4000_Hex) OTE(MCC3_18G_CommsOK) ,E300ToMotor(AOI_MCC3_18G_ToPLC1,MotorsStatusTag.MCC3_18G,AOP_MCC3_18G:I,MCC3_18G_CommsOK) ];
   188: [GSV(Module,AOP_MCC3_18J,EntryStatus,GSV_EntryStatus) MEQ(GSV_EntryStatus,16#f000,Const_4000_Hex) OTE(MCC3_18J_CommsOK) ,E300ToMotor(AOI_MCC3_18J_ToPLC1,MotorsStatusTag.MCC3_18J,AOP_MCC3_18J:I,MCC3_18J_CommsOK) ];
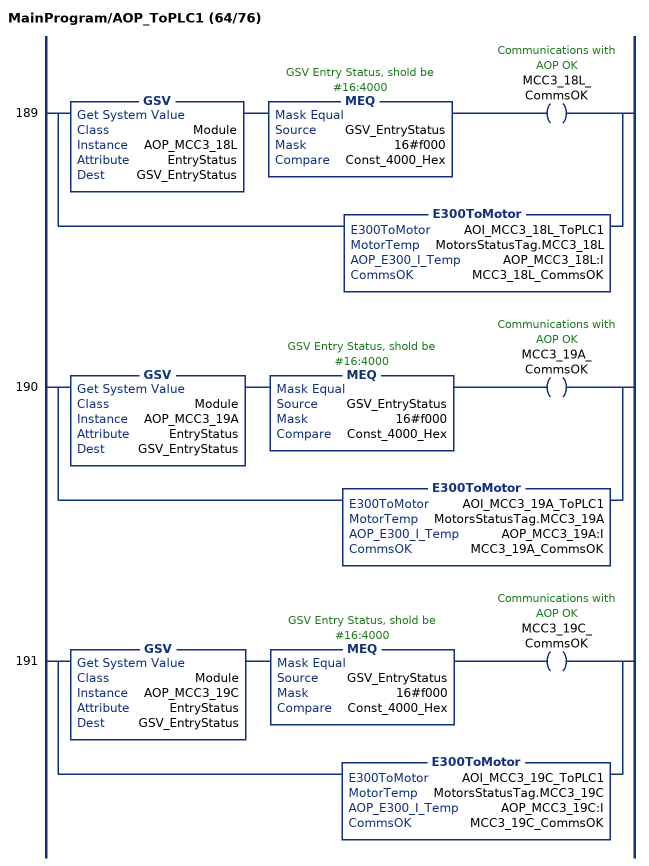
   189: [GSV(Module,AOP_MCC3_18L,EntryStatus,GSV_EntryStatus) MEQ(GSV_EntryStatus,16#f000,Const_4000_Hex) OTE(MCC3_18L_CommsOK) ,E300ToMotor(AOI_MCC3_18L_ToPLC1,MotorsStatusTag.MCC3_18L,AOP_MCC3_18L:I,MCC3_18L_CommsOK) ];
   190: [GSV(Module,AOP_MCC3_19A,EntryStatus,GSV_EntryStatus) MEQ(GSV_EntryStatus,16#f000,Const_4000_Hex) OTE(MCC3_19A_CommsOK) ,E300ToMotor(AOI_MCC3_19A_ToPLC1,MotorsStatusTag.MCC3_19A,AOP_MCC3_19A:I,MCC3_19A_CommsOK) ];
   191: [GSV(Module,AOP_MCC3_19C,EntryStatus,GSV_EntryStatus) MEQ(GSV_EntryStatus,16#f000,Const_4000_Hex) OTE(MCC3_19C_CommsOK) ,E300ToMotor(AOI_MCC3_19C_ToPLC1,MotorsStatusTag.MCC3_19C,AOP_MCC3_19C:I,MCC3_19C_CommsOK) ];
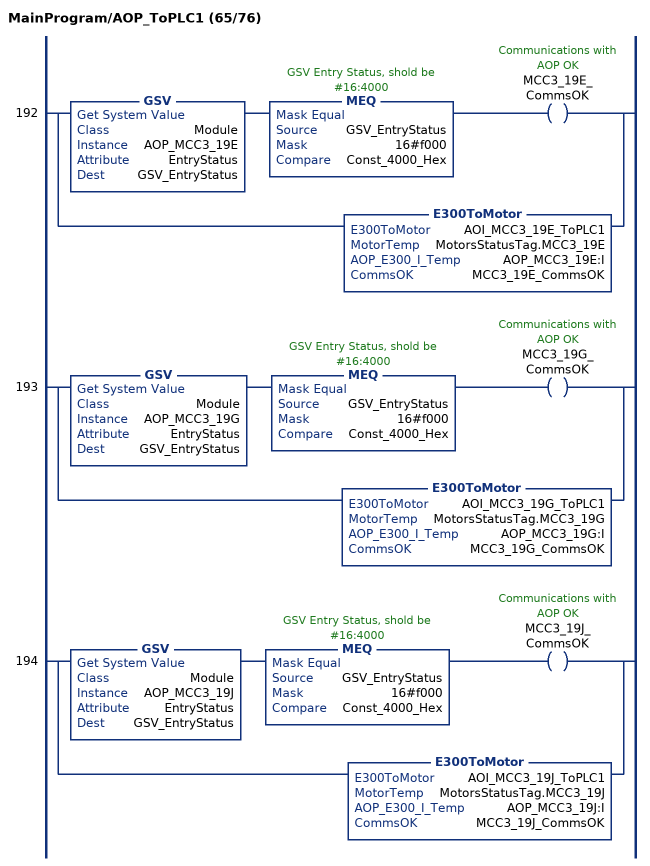
   192: [GSV(Module,AOP_MCC3_19E,EntryStatus,GSV_EntryStatus) MEQ(GSV_EntryStatus,16#f000,Const_4000_Hex) OTE(MCC3_19E_CommsOK) ,E300ToMotor(AOI_MCC3_19E_ToPLC1,MotorsStatusTag.MCC3_19E,AOP_MCC3_19E:I,MCC3_19E_CommsOK) ];
   193: [GSV(Module,AOP_MCC3_19G,EntryStatus,GSV_EntryStatus) MEQ(GSV_EntryStatus,16#f000,Const_4000_Hex) OTE(MCC3_19G_CommsOK) ,E300ToMotor(AOI_MCC3_19G_ToPLC1,MotorsStatusTag.MCC3_19G,AOP_MCC3_19G:I,MCC3_19G_CommsOK) ];
   194: [GSV(Module,AOP_MCC3_19J,EntryStatus,GSV_EntryStatus) MEQ(GSV_EntryStatus,16#f000,Const_4000_Hex) OTE(MCC3_19J_CommsOK) ,E300ToMotor(AOI_MCC3_19J_ToPLC1,MotorsStatusTag.MCC3_19J,AOP_MCC3_19J:I,MCC3_19J_CommsOK) ];
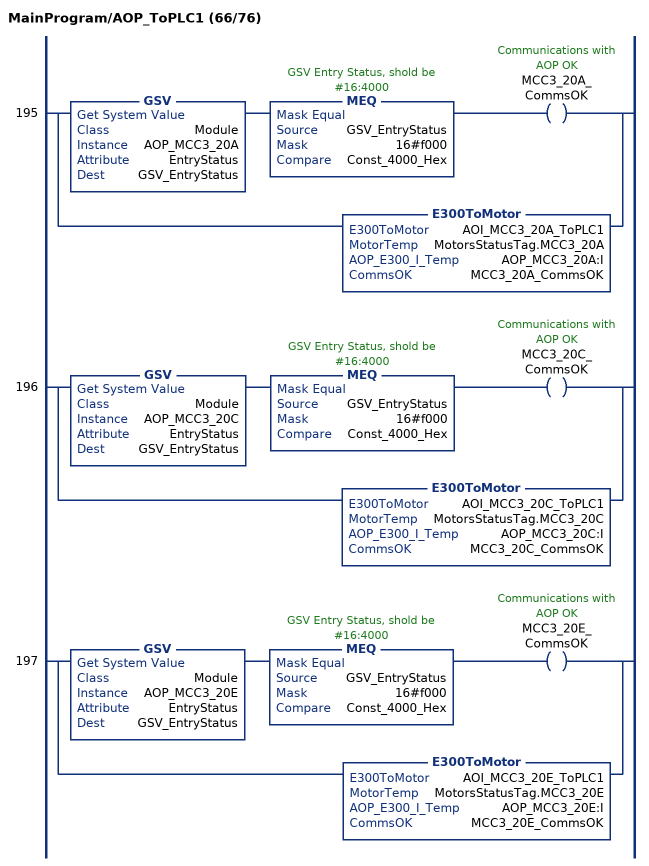
   195: [GSV(Module,AOP_MCC3_20A,EntryStatus,GSV_EntryStatus) MEQ(GSV_EntryStatus,16#f000,Const_4000_Hex) OTE(MCC3_20A_CommsOK) ,E300ToMotor(AOI_MCC3_20A_ToPLC1,MotorsStatusTag.MCC3_20A,AOP_MCC3_20A:I,MCC3_20A_CommsOK) ];
   196: [GSV(Module,AOP_MCC3_20C,EntryStatus,GSV_EntryStatus) MEQ(GSV_EntryStatus,16#f000,Const_4000_Hex) OTE(MCC3_20C_CommsOK) ,E300ToMotor(AOI_MCC3_20C_ToPLC1,MotorsStatusTag.MCC3_20C,AOP_MCC3_20C:I,MCC3_20C_CommsOK) ];
   197: [GSV(Module,AOP_MCC3_20E,EntryStatus,GSV_EntryStatus) MEQ(GSV_EntryStatus,16#f000,Const_4000_Hex) OTE(MCC3_20E_CommsOK) ,E300ToMotor(AOI_MCC3_20E_ToPLC1,MotorsStatusTag.MCC3_20E,AOP_MCC3_20E:I,MCC3_20E_CommsOK) ];
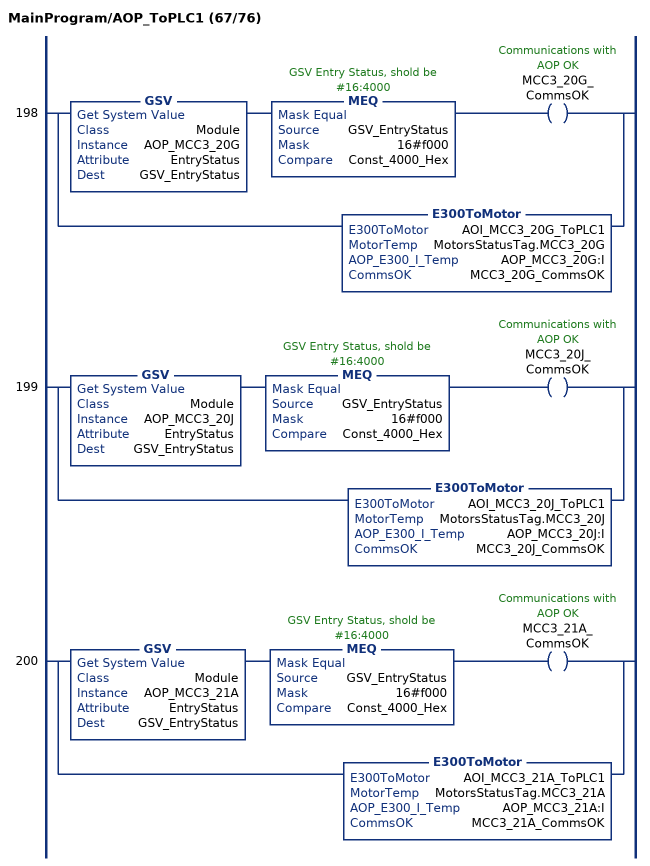
   198: [GSV(Module,AOP_MCC3_20G,EntryStatus,GSV_EntryStatus) MEQ(GSV_EntryStatus,16#f000,Const_4000_Hex) OTE(MCC3_20G_CommsOK) ,E300ToMotor(AOI_MCC3_20G_ToPLC1,MotorsStatusTag.MCC3_20G,AOP_MCC3_20G:I,MCC3_20G_CommsOK) ];
   199: [GSV(Module,AOP_MCC3_20J,EntryStatus,GSV_EntryStatus) MEQ(GSV_EntryStatus,16#f000,Const_4000_Hex) OTE(MCC3_20J_CommsOK) ,E300ToMotor(AOI_MCC3_20J_ToPLC1,MotorsStatusTag.MCC3_20J,AOP_MCC3_20J:I,MCC3_20J_CommsOK) ];
   200: [GSV(Module,AOP_MCC3_21A,EntryStatus,GSV_EntryStatus) MEQ(GSV_EntryStatus,16#f000,Const_4000_Hex) OTE(MCC3_21A_CommsOK) ,E300ToMotor(AOI_MCC3_21A_ToPLC1,MotorsStatusTag.MCC3_21A,AOP_MCC3_21A:I,MCC3_21A_CommsOK) ];
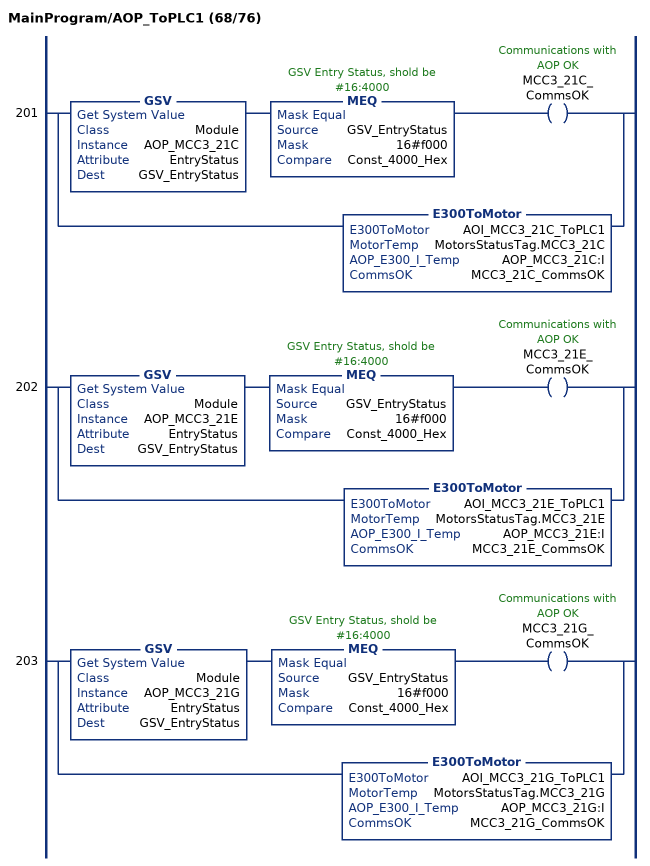
   201: [GSV(Module,AOP_MCC3_21C,EntryStatus,GSV_EntryStatus) MEQ(GSV_EntryStatus,16#f000,Const_4000_Hex) OTE(MCC3_21C_CommsOK) ,E300ToMotor(AOI_MCC3_21C_ToPLC1,MotorsStatusTag.MCC3_21C,AOP_MCC3_21C:I,MCC3_21C_CommsOK) ];
   202: [GSV(Module,AOP_MCC3_21E,EntryStatus,GSV_EntryStatus) MEQ(GSV_EntryStatus,16#f000,Const_4000_Hex) OTE(MCC3_21E_CommsOK) ,E300ToMotor(AOI_MCC3_21E_ToPLC1,MotorsStatusTag.MCC3_21E,AOP_MCC3_21E:I,MCC3_21E_CommsOK) ];
   203: [GSV(Module,AOP_MCC3_21G,EntryStatus,GSV_EntryStatus) MEQ(GSV_EntryStatus,16#f000,Const_4000_Hex) OTE(MCC3_21G_CommsOK) ,E300ToMotor(AOI_MCC3_21G_ToPLC1,MotorsStatusTag.MCC3_21G,AOP_MCC3_21G:I,MCC3_21G_CommsOK) ];
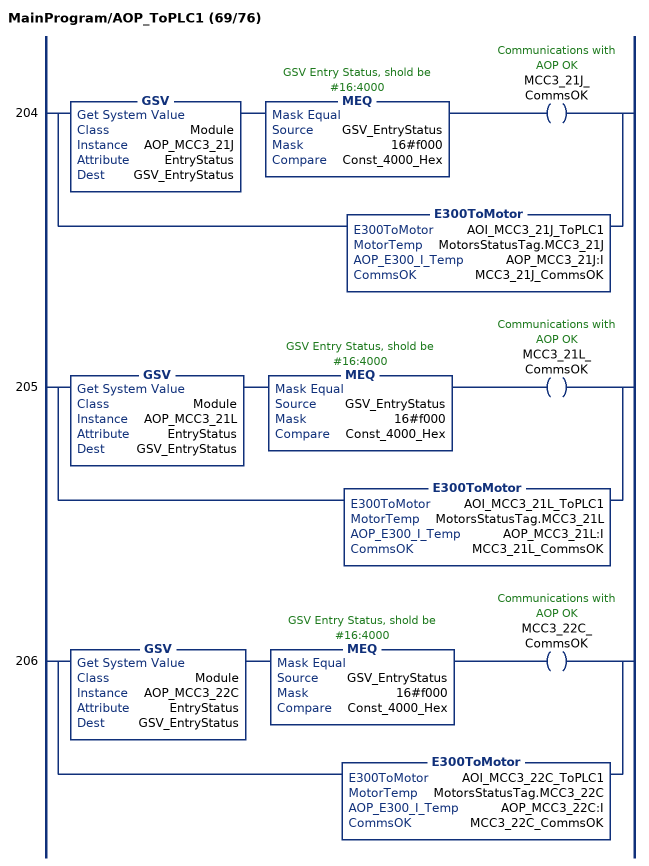
   204: [GSV(Module,AOP_MCC3_21J,EntryStatus,GSV_EntryStatus) MEQ(GSV_EntryStatus,16#f000,Const_4000_Hex) OTE(MCC3_21J_CommsOK) ,E300ToMotor(AOI_MCC3_21J_ToPLC1,MotorsStatusTag.MCC3_21J,AOP_MCC3_21J:I,MCC3_21J_CommsOK) ];
   205: [GSV(Module,AOP_MCC3_21L,EntryStatus,GSV_EntryStatus) MEQ(GSV_EntryStatus,16#f000,Const_4000_Hex) OTE(MCC3_21L_CommsOK) ,E300ToMotor(AOI_MCC3_21L_ToPLC1,MotorsStatusTag.MCC3_21L,AOP_MCC3_21L:I,MCC3_21L_CommsOK) ];
   206: [GSV(Module,AOP_MCC3_22C,EntryStatus,GSV_EntryStatus) MEQ(GSV_EntryStatus,16#f000,Const_4000_Hex) OTE(MCC3_22C_CommsOK) ,E300ToMotor(AOI_MCC3_22C_ToPLC1,MotorsStatusTag.MCC3_22C,AOP_MCC3_22C:I,MCC3_22C_CommsOK) ];
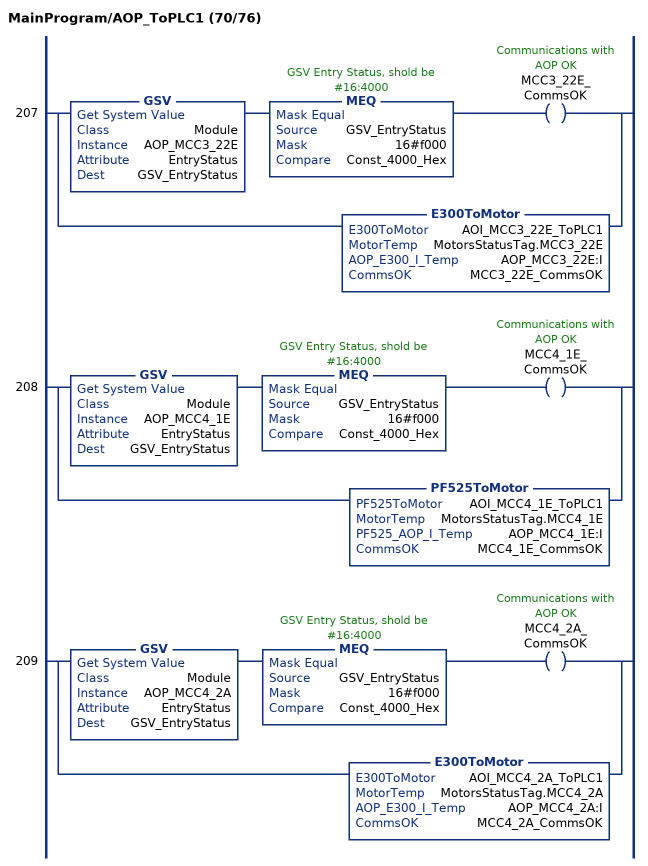
   207: [GSV(Module,AOP_MCC3_22E,EntryStatus,GSV_EntryStatus) MEQ(GSV_EntryStatus,16#f000,Const_4000_Hex) OTE(MCC3_22E_CommsOK) ,E300ToMotor(AOI_MCC3_22E_ToPLC1,MotorsStatusTag.MCC3_22E,AOP_MCC3_22E:I,MCC3_22E_CommsOK) ];
   208: [GSV(Module,AOP_MCC4_1E,EntryStatus,GSV_EntryStatus) MEQ(GSV_EntryStatus,16#f000,Const_4000_Hex) OTE(MCC4_1E_CommsOK) ,PF525ToMotor(AOI_MCC4_1E_ToPLC1,MotorsStatusTag.MCC4_1E,AOP_MCC4_1E:I,MCC4_1E_CommsOK) ];
   209: [GSV(Module,AOP_MCC4_2A,EntryStatus,GSV_EntryStatus) MEQ(GSV_EntryStatus,16#f000,Const_4000_Hex) OTE(MCC4_2A_CommsOK) ,E300ToMotor(AOI_MCC4_2A_ToPLC1,MotorsStatusTag.MCC4_2A,AOP_MCC4_2A:I,MCC4_2A_CommsOK) ];
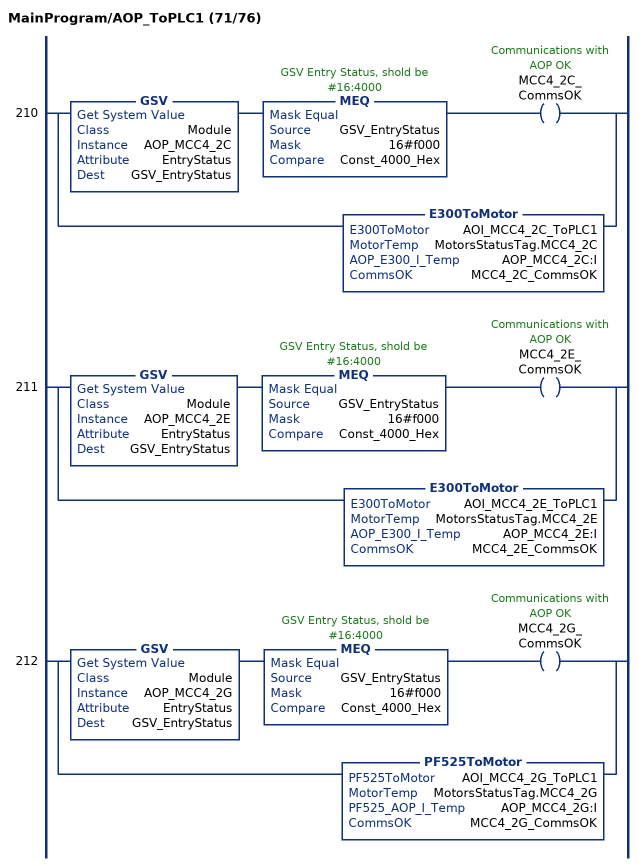
   210: [GSV(Module,AOP_MCC4_2C,EntryStatus,GSV_EntryStatus) MEQ(GSV_EntryStatus,16#f000,Const_4000_Hex) OTE(MCC4_2C_CommsOK) ,E300ToMotor(AOI_MCC4_2C_ToPLC1,MotorsStatusTag.MCC4_2C,AOP_MCC4_2C:I,MCC4_2C_CommsOK) ];
   211: [GSV(Module,AOP_MCC4_2E,EntryStatus,GSV_EntryStatus) MEQ(GSV_EntryStatus,16#f000,Const_4000_Hex) OTE(MCC4_2E_CommsOK) ,E300ToMotor(AOI_MCC4_2E_ToPLC1,MotorsStatusTag.MCC4_2E,AOP_MCC4_2E:I,MCC4_2E_CommsOK) ];
   212: [GSV(Module,AOP_MCC4_2G,EntryStatus,GSV_EntryStatus) MEQ(GSV_EntryStatus,16#f000,Const_4000_Hex) OTE(MCC4_2G_CommsOK) ,PF525ToMotor(AOI_MCC4_2G_ToPLC1,MotorsStatusTag.MCC4_2G,AOP_MCC4_2G:I,MCC4_2G_CommsOK) ];
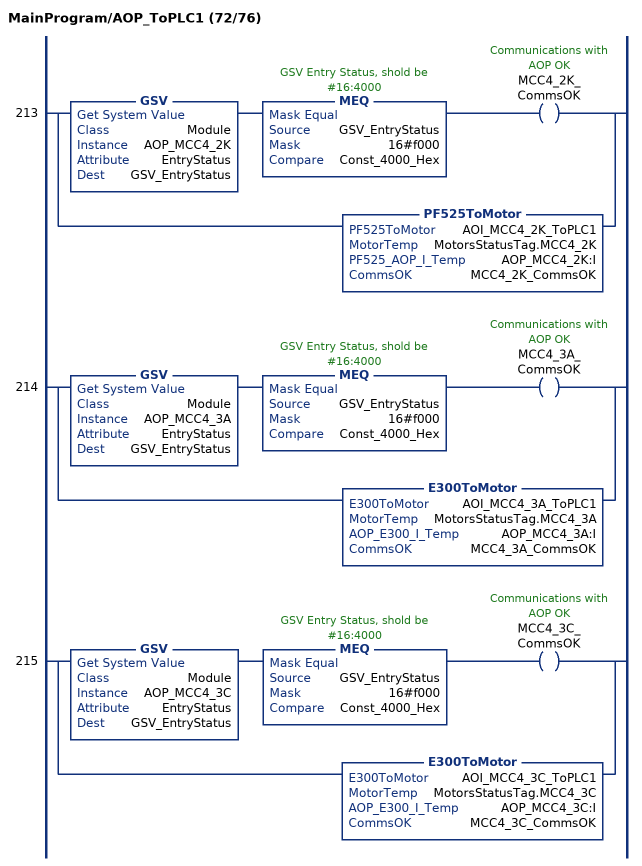
   213: [GSV(Module,AOP_MCC4_2K,EntryStatus,GSV_EntryStatus) MEQ(GSV_EntryStatus,16#f000,Const_4000_Hex) OTE(MCC4_2K_CommsOK) ,PF525ToMotor(AOI_MCC4_2K_ToPLC1,MotorsStatusTag.MCC4_2K,AOP_MCC4_2K:I,MCC4_2K_CommsOK) ];
   214: [GSV(Module,AOP_MCC4_3A,EntryStatus,GSV_EntryStatus) MEQ(GSV_EntryStatus,16#f000,Const_4000_Hex) OTE(MCC4_3A_CommsOK) ,E300ToMotor(AOI_MCC4_3A_ToPLC1,MotorsStatusTag.MCC4_3A,AOP_MCC4_3A:I,MCC4_3A_CommsOK) ];
   215: [GSV(Module,AOP_MCC4_3C,EntryStatus,GSV_EntryStatus) MEQ(GSV_EntryStatus,16#f000,Const_4000_Hex) OTE(MCC4_3C_CommsOK) ,E300ToMotor(AOI_MCC4_3C_ToPLC1,MotorsStatusTag.MCC4_3C,AOP_MCC4_3C:I,MCC4_3C_CommsOK) ];
